{attribute 'qualified_only'}
{attribute 'strict'}
TYPE E_CncServoCommand :
(
	NoCommand,
	Base,
	MovePos,
	Fixed,
	Release
);
END_TYPE

(* stored: Version 1.1.0.1, ProductVersion 3.1.4024.12
   EnumerationTextList E_CncServoCommand: Id {6a8c5627-479c-4fb0-b798-28bdec7d6b55} *)
